TYPE ST_OutputStationHSCurrentConfigurationGeneral :
STRUCT
	{attribute 'OPC.UA.DA.Description' := 'Dummy (for making struct visible on OPC UA'}
	Dummy						: BOOL;
END_STRUCT
END_TYPE

(* stored: Version 1.1.0.1, ProductVersion 3.1.4024.2
   DUT ST_OutputStationHSCurrentConfigurationGeneral: Id {aa989f3c-d5c6-488b-baf4-9f61913f5bed} *)
